
// ===== library: MasterCopy "FB_SingleSolCyl_LAD" =====

// folder: FB_SingleSolenoidCylinder

FUNCTION_BLOCK "FB_SingleSolCyl_LAD"   // FB2103, LAD
{ S7_Optimized_Access := 'TRUE' }
   VAR_INPUT
      Enable : Bool := 1;   // 使能单控气缸控制块，FALSE时关闭输出并禁止动作
      Mode : Int;   // 模式选择：1=Manual手动，2=Auto自动；其它值报警
      Exe_Auto : Bool;   // 自动模式下的动作命令，1伸出，0缩回
      Exe_Manual : Bool;   // 手动模式下的动作命令，1伸出，0缩回
      Sensor_Ext : Bool;   // 气缸伸出到位检测信号
      Sensor_Home : Bool;   // 气缸缩回原点检测信号
      Reset : Bool;   // 报警复位命令，清除报警和报警代码
      Timeout : Time := T#3S;   // 伸出或缩回等待传感器到位的超时时间，例如T#5s
   END_VAR
   VAR_OUTPUT
      Q : Bool;   // 控制真实电磁阀Q点，TRUE气缸伸出，FALSE气缸缩回
      Error : Bool;   // 报警锁存输出，需要ResetAlarm清除
      Error_Status : Word;   // 报警代码：2模式无效，3传感器冲突，257伸出超时，258缩回超时
      Extend : Bool;   // 当前有效模式下的伸出命令
      Retract : Bool;   // 当前有效模式下的缩回命令
      AutoActive : Bool;   // 自动模式有效状态：Enable、Mode=2、无报警
      ManualActive : Bool;   // 手动模式有效状态：Enable、Mode=1、无报警
   END_VAR
   VAR
      ExtendTimeoutTimer : TON_TIME;   // 伸出动作超时TON实例
      RetractTimeoutTimer : TON_TIME;   // 缩回动作超时TON实例
   END_VAR
   VAR_TEMP   // added for the SCL form of the ladder/FBD networks
      _w1 : Bool;
   END_VAR
BEGIN

REGION Network 1: 报警复位
   // ResetAlarm时清除报警锁存和报警代码。
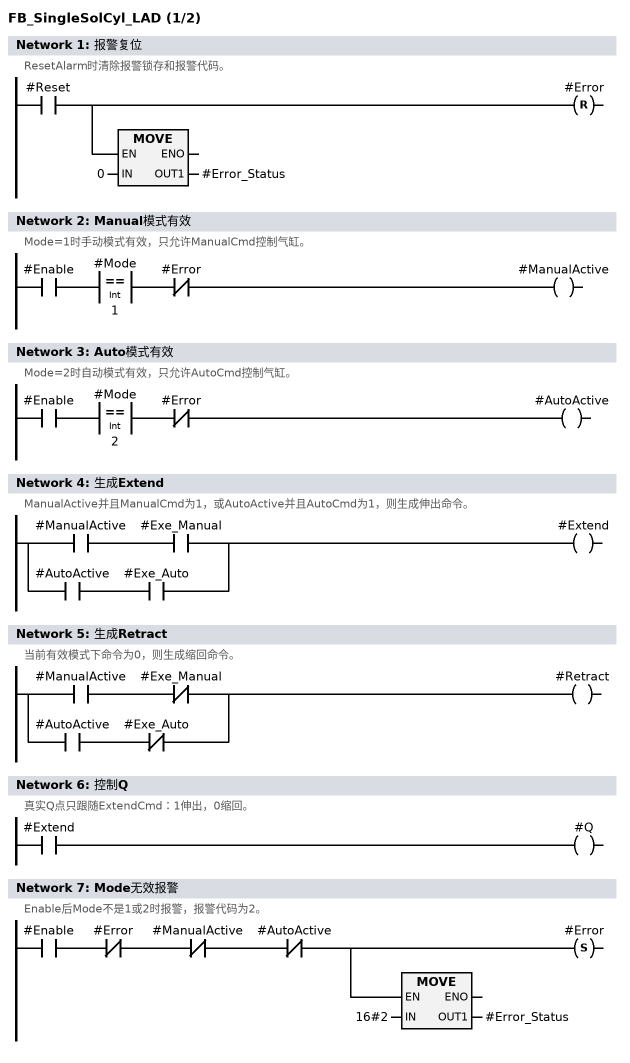
   RUNG wire#powerrail
      Contact( #Reset )
      wire#w1
      R_Coil( #Error )
   END_RUNG
   RUNG wire#w1
      { S7_GenerateENO := "TRUE" } Move(in := 0, out1 => #Error_Status)
   END_RUNG
   // the same network as SCL:
   IF #Reset THEN
       #Error := FALSE;
       #Error_Status := 0;
   END_IF;
END_REGION

REGION Network 2: Manual模式有效
   // Mode=1时手动模式有效，只允许ManualCmd控制气缸。
   RUNG wire#powerrail
      Contact( #Enable )
      { S7_Templates := "SrcType := Int" } EQ_Contact(in1 := #Mode, in2 := 1)
      I_Contact( #Error )
      Coil( #ManualActive )
   END_RUNG
   // the same network as SCL:
   #ManualActive := #Enable AND (#Mode = 1) AND NOT #Error;
END_REGION

REGION Network 3: Auto模式有效
   // Mode=2时自动模式有效，只允许AutoCmd控制气缸。
   RUNG wire#powerrail
      Contact( #Enable )
      { S7_Templates := "SrcType := Int" } EQ_Contact(in1 := #Mode, in2 := 2)
      I_Contact( #Error )
      Coil( #AutoActive )
   END_RUNG
   // the same network as SCL:
   #AutoActive := #Enable AND (#Mode = 2) AND NOT #Error;
END_REGION

REGION Network 4: 生成Extend
   // ManualActive并且ManualCmd为1，或AutoActive并且AutoCmd为1，则生成伸出命令。
   RUNG wire#powerrail
      Contact( #ManualActive )
      Contact( #Exe_Manual )
      wire#w1
      Coil( #Extend )
   END_RUNG
   RUNG wire#powerrail
      Contact( #AutoActive )
      Contact( #Exe_Auto )
   END_RUNG wire#w1
   // the same network as SCL:
   #Extend := (#ManualActive AND #Exe_Manual) OR (#AutoActive AND #Exe_Auto);
END_REGION

REGION Network 5: 生成Retract
   // 当前有效模式下命令为0，则生成缩回命令。
   RUNG wire#powerrail
      Contact( #ManualActive )
      I_Contact( #Exe_Manual )
      wire#w1
      Coil( #Retract )
   END_RUNG
   RUNG wire#powerrail
      Contact( #AutoActive )
      I_Contact( #Exe_Auto )
   END_RUNG wire#w1
   // the same network as SCL:
   #Retract := (#ManualActive AND NOT #Exe_Manual) OR (#AutoActive AND NOT #Exe_Auto);
END_REGION

REGION Network 6: 控制Q
   // 真实Q点只跟随ExtendCmd：1伸出，0缩回。
   RUNG wire#powerrail
      Contact( #Extend )
      Coil( #Q )
   END_RUNG
   // the same network as SCL:
   #Q := #Extend;
END_REGION

REGION Network 7: Mode无效报警
   // Enable后Mode不是1或2时报警，报警代码为2。
   RUNG wire#powerrail
      Contact( #Enable )
      I_Contact( #Error )
      I_Contact( #ManualActive )
      I_Contact( #AutoActive )
      wire#w1
      S_Coil( #Error )
   END_RUNG
   RUNG wire#w1
      { S7_GenerateENO := "TRUE" } Move(in := 16#2, out1 => #Error_Status)
   END_RUNG
   // the same network as SCL:
   #_w1 := #Enable AND NOT #Error AND NOT #ManualActive AND NOT #AutoActive;
   IF #_w1 THEN
       #Error := TRUE;
       #Error_Status := 16#2;
   END_IF;
END_REGION

REGION Network 8: 传感器冲突报警
   // 伸出到位和缩回原点不能同时为1。
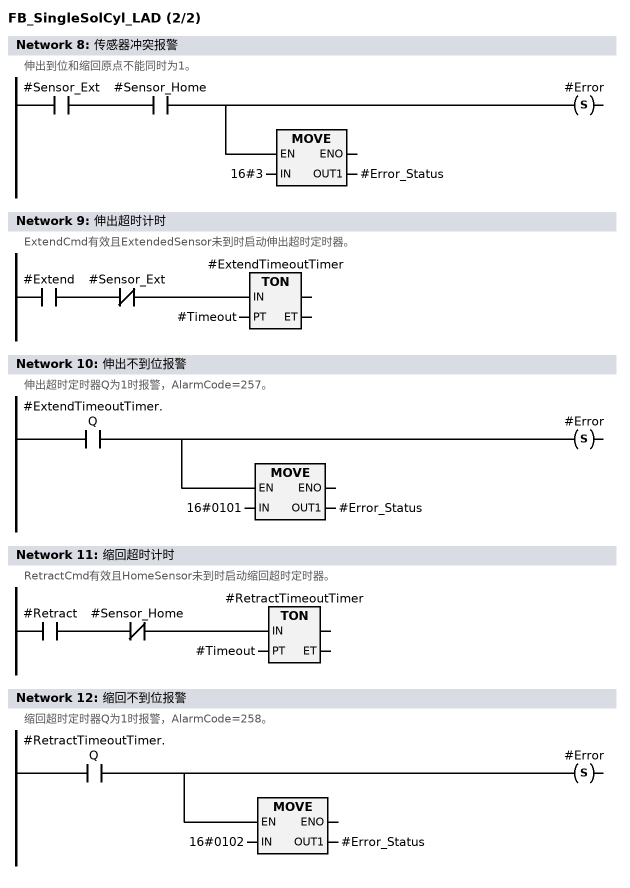
   RUNG wire#powerrail
      Contact( #Sensor_Ext )
      Contact( #Sensor_Home )
      wire#w1
      S_Coil( #Error )
   END_RUNG
   RUNG wire#w1
      { S7_GenerateENO := "TRUE" } Move(in := 16#3, out1 => #Error_Status)
   END_RUNG
   // the same network as SCL:
   IF #Sensor_Ext AND #Sensor_Home THEN
       #Error := TRUE;
       #Error_Status := 16#3;
   END_IF;
END_REGION

REGION Network 9: 伸出超时计时
   // ExtendCmd有效且ExtendedSensor未到时启动伸出超时定时器。
   #ExtendTimeoutTimer(IN := #Extend AND NOT #Sensor_Ext, PT := #Timeout);   // TON
END_REGION

REGION Network 10: 伸出不到位报警
   // 伸出超时定时器Q为1时报警，AlarmCode=257。
   RUNG wire#powerrail
      Contact( #ExtendTimeoutTimer.Q )
      wire#w1
      S_Coil( #Error )
   END_RUNG
   RUNG wire#w1
      { S7_GenerateENO := "TRUE" } Move(in := 16#0101, out1 => #Error_Status)
   END_RUNG
   // the same network as SCL:
   IF #ExtendTimeoutTimer.Q THEN
       #Error := TRUE;
       #Error_Status := 16#0101;
   END_IF;
END_REGION

REGION Network 11: 缩回超时计时
   // RetractCmd有效且HomeSensor未到时启动缩回超时定时器。
   #RetractTimeoutTimer(IN := #Retract AND NOT #Sensor_Home, PT := #Timeout);   // TON
END_REGION

REGION Network 12: 缩回不到位报警
   // 缩回超时定时器Q为1时报警，AlarmCode=258。
   RUNG wire#powerrail
      Contact( #RetractTimeoutTimer.Q )
      wire#w1
      S_Coil( #Error )
   END_RUNG
   RUNG wire#w1
      { S7_GenerateENO := "TRUE" } Move(in := 16#0102, out1 => #Error_Status)
   END_RUNG
   // the same network as SCL:
   IF #RetractTimeoutTimer.Q THEN
       #Error := TRUE;
       #Error_Status := 16#0102;
   END_IF;
END_REGION
END_FUNCTION_BLOCK

// ===== library: MasterCopy "FB_SingleSolCyl_SCL" =====

// folder: FB_SingleSolenoidCylinder

FUNCTION_BLOCK "FB_SingleSolCyl_SCL"   // FB2104, LAD
{ S7_Optimized_Access := 'TRUE' }
   VAR_INPUT
      Enable : Bool := 1;   // 使能单控气缸控制块，FALSE时关闭输出并禁止动作
      Mode : Int;   // 模式选择：1=Manual手动，2=Auto自动；其它值报警
      Exe_Auto : Bool;   // 自动模式下的动作命令，1伸出，0缩回
      Exe_Manual : Bool;   // 手动模式下的动作命令，1伸出，0缩回
      Sensor_Ext : Bool;   // 气缸伸出到位检测信号
      Sensor_Home : Bool;   // 气缸缩回原点检测信号
      Reset : Bool;   // 报警复位命令，清除报警和报警代码
      Timeout : Time := T#3S;   // 伸出或缩回等待传感器到位的超时时间，例如T#5s
   END_VAR
   VAR_OUTPUT
      Q : Bool;   // 控制真实电磁阀Q点，TRUE气缸伸出，FALSE气缸缩回
      Error : Bool;   // 报警锁存输出，需要ResetAlarm清除
      Error_Status : Word;   // 报警代码：2模式无效，3传感器冲突，257伸出超时，258缩回超时
      Extend : Bool;   // 当前有效模式下的伸出命令
      Retract : Bool;   // 当前有效模式下的缩回命令
      AutoActive : Bool;   // 自动模式有效状态：Enable、Mode=2、无报警
      ManualActive : Bool;   // 手动模式有效状态：Enable、Mode=1、无报警
   END_VAR
   VAR
      ExtendTimeoutTimer : TON_TIME;   // 伸出动作超时TON实例
      RetractTimeoutTimer : TON_TIME;   // 缩回动作超时TON实例
   END_VAR
BEGIN

REGION Network 1 (SCL): 条件判断集中处理
   // 报警、动作命令、伸出/缩回超时集中在本SCL程序段处理；ManualActive、AutoActive和Q输出保留LAD程序段。
   // 条件集中处理：报警、命令、超时都放在本SCL程序段
   // 保留LAD程序段只负责：ManualActive、AutoActive、Q输出

   // Reset优先清除报警；若故障原因仍存在，后续逻辑会重新报警
   IF #Reset THEN
       #Error := FALSE;
       #Error_Status := W#16#0000;
   END_IF;

   // 默认先清除动作命令，避免无效模式或报警时误动作
   #Extend := FALSE;
   #Retract := FALSE;

   // 根据有效模式生成动作命令：1伸出，0缩回
   IF #Enable AND NOT #Error THEN
       IF #ManualActive THEN
           #Extend := #Exe_Manual;
           #Retract := NOT #Exe_Manual;
       ELSIF #AutoActive THEN
           #Extend := #Exe_Auto;
           #Retract := NOT #Exe_Auto;
       END_IF;
   END_IF;

   // 定时器集中调用：伸出等待Sensor_Ext，缩回等待Sensor_Home
   #ExtendTimeoutTimer(IN := #Extend AND NOT #Sensor_Ext,
                       PT := #Timeout);
   #RetractTimeoutTimer(IN := #Retract AND NOT #Sensor_Home,
                        PT := #Timeout);

   // 报警判断集中处理
   IF #Enable AND NOT #Error THEN
       // Mode只能为1或2；
       IF (#Mode <> 1) AND (#Mode <> 2) THEN
           #Error := TRUE;
           #Error_Status := W#16#0002;

       // 两个极限传感器不能同时为1
       ELSIF #Sensor_Ext AND #Sensor_Home THEN
           #Error := TRUE;
           #Error_Status := W#16#0003;

       // 伸出不到位超时
       ELSIF #ExtendTimeoutTimer.Q THEN
           #Error := TRUE;
           #Error_Status := W#16#0101;

       // 缩回不到位超时
       ELSIF #RetractTimeoutTimer.Q THEN
           #Error := TRUE;
           #Error_Status := W#16#0102;
       END_IF;
   END_IF;

   // 报警后本扫描周期立即撤销有效模式和动作命令，后续LAD Q输出保持安全关闭
   IF #Error THEN
       #ManualActive := FALSE;
       #AutoActive := FALSE;
       #Extend := FALSE;
       #Retract := FALSE;
   END_IF;
END_REGION

REGION Network 2: Manual模式有效
   // Mode=1时手动模式有效，只允许ManualCmd控制气缸。
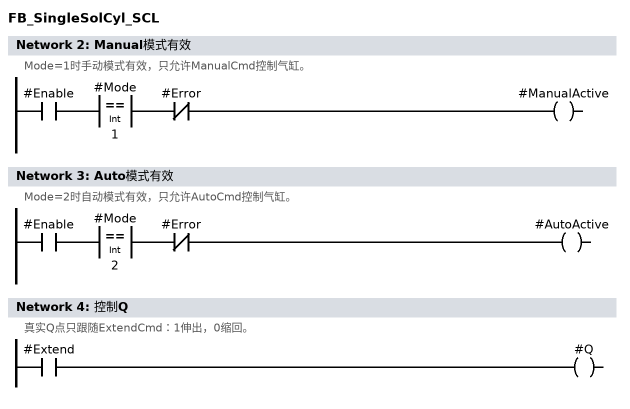
   RUNG wire#powerrail
      Contact( #Enable )
      { S7_Templates := "SrcType := Int" } EQ_Contact(in1 := #Mode, in2 := 1)
      I_Contact( #Error )
      Coil( #ManualActive )
   END_RUNG
   // the same network as SCL:
   #ManualActive := #Enable AND (#Mode = 1) AND NOT #Error;
END_REGION

REGION Network 3: Auto模式有效
   // Mode=2时自动模式有效，只允许AutoCmd控制气缸。
   RUNG wire#powerrail
      Contact( #Enable )
      { S7_Templates := "SrcType := Int" } EQ_Contact(in1 := #Mode, in2 := 2)
      I_Contact( #Error )
      Coil( #AutoActive )
   END_RUNG
   // the same network as SCL:
   #AutoActive := #Enable AND (#Mode = 2) AND NOT #Error;
END_REGION

REGION Network 4: 控制Q
   // 真实Q点只跟随ExtendCmd：1伸出，0缩回。
   RUNG wire#powerrail
      Contact( #Extend )
      Coil( #Q )
   END_RUNG
   // the same network as SCL:
   #Q := #Extend;
END_REGION
END_FUNCTION_BLOCK